Staubli VAL3: CMS_Module.dtx

bool bDoAirex = true
bool bGlueGlass
public dio doJ206_EtherCAT_Box_1__CPX_FB37__Q0 = {link=J206_EtherCAT\Box_1_(CPX-FB37)\%Q0}
public dio doJ206_EtherCAT_Box_1__CPX_FB37__Q1 = {link=J206_EtherCAT\Box_1_(CPX-FB37)\%Q1}
public dio doJ206_EtherCAT_Box_1__CPX_FB37__Q10 = {link=J206_EtherCAT\Box_1_(CPX-FB37)\%Q10}
public dio doJ206_EtherCAT_Box_1__CPX_FB37__Q11 = {link=J206_EtherCAT\Box_1_(CPX-FB37)\%Q11}
public dio doJ206_EtherCAT_Box_1__CPX_FB37__Q12 = {link=J206_EtherCAT\Box_1_(CPX-FB37)\%Q12}
public dio doJ206_EtherCAT_Box_1__CPX_FB37__Q13 = {link=J206_EtherCAT\Box_1_(CPX-FB37)\%Q13}
public dio doJ206_EtherCAT_Box_1__CPX_FB37__Q14 = {link=J206_EtherCAT\Box_1_(CPX-FB37)\%Q14}
public dio doJ206_EtherCAT_Box_1__CPX_FB37__Q15 = {link=J206_EtherCAT\Box_1_(CPX-FB37)\%Q15}
public dio doJ206_EtherCAT_Box_1__CPX_FB37__Q16 = {link=J206_EtherCAT\Box_1_(CPX-FB37)\%Q16}
public dio doJ206_EtherCAT_Box_1__CPX_FB37__Q17 = {link=J206_EtherCAT\Box_1_(CPX-FB37)\%Q17}
public dio doJ206_EtherCAT_Box_1__CPX_FB37__Q18 = {link=J206_EtherCAT\Box_1_(CPX-FB37)\%Q18}
public dio doJ206_EtherCAT_Box_1__CPX_FB37__Q19 = {link=J206_EtherCAT\Box_1_(CPX-FB37)\%Q19}
public dio doJ206_EtherCAT_Box_1__CPX_FB37__Q2 = {link=J206_EtherCAT\Box_1_(CPX-FB37)\%Q2}
public dio doJ206_EtherCAT_Box_1__CPX_FB37__Q20 = {link=J206_EtherCAT\Box_1_(CPX-FB37)\%Q20}
public dio doJ206_EtherCAT_Box_1__CPX_FB37__Q21 = {link=J206_EtherCAT\Box_1_(CPX-FB37)\%Q21}
public dio doJ206_EtherCAT_Box_1__CPX_FB37__Q22 = {link=J206_EtherCAT\Box_1_(CPX-FB37)\%Q22}
public dio doJ206_EtherCAT_Box_1__CPX_FB37__Q23 = {link=J206_EtherCAT\Box_1_(CPX-FB37)\%Q23}
public dio doJ206_EtherCAT_Box_1__CPX_FB37__Q24 = {link=J206_EtherCAT\Box_1_(CPX-FB37)\%Q24}
public dio doJ206_EtherCAT_Box_1__CPX_FB37__Q25 = {link=J206_EtherCAT\Box_1_(CPX-FB37)\%Q25}
public dio doJ206_EtherCAT_Box_1__CPX_FB37__Q26 = {link=J206_EtherCAT\Box_1_(CPX-FB37)\%Q26}
public dio doJ206_EtherCAT_Box_1__CPX_FB37__Q27 = {link=J206_EtherCAT\Box_1_(CPX-FB37)\%Q27}
public dio doJ206_EtherCAT_Box_1__CPX_FB37__Q28 = {link=J206_EtherCAT\Box_1_(CPX-FB37)\%Q28}
public dio doJ206_EtherCAT_Box_1__CPX_FB37__Q29 = {link=J206_EtherCAT\Box_1_(CPX-FB37)\%Q29}
public dio doJ206_EtherCAT_Box_1__CPX_FB37__Q3 = {link=J206_EtherCAT\Box_1_(CPX-FB37)\%Q3}
public dio doJ206_EtherCAT_Box_1__CPX_FB37__Q30 = {link=J206_EtherCAT\Box_1_(CPX-FB37)\%Q30}
public dio doJ206_EtherCAT_Box_1__CPX_FB37__Q31 = {link=J206_EtherCAT\Box_1_(CPX-FB37)\%Q31}
public dio doJ206_EtherCAT_Box_1__CPX_FB37__Q4 = {link=J206_EtherCAT\Box_1_(CPX-FB37)\%Q4}
public dio doJ206_EtherCAT_Box_1__CPX_FB37__Q5 = {link=J206_EtherCAT\Box_1_(CPX-FB37)\%Q5}
public dio doJ206_EtherCAT_Box_1__CPX_FB37__Q6 = {link=J206_EtherCAT\Box_1_(CPX-FB37)\%Q6}
public dio doJ206_EtherCAT_Box_1__CPX_FB37__Q7 = {link=J206_EtherCAT\Box_1_(CPX-FB37)\%Q7}
public dio doJ206_EtherCAT_Box_1__CPX_FB37__Q8 = {link=J206_EtherCAT\Box_1_(CPX-FB37)\%Q8}
public dio doJ206_EtherCAT_Box_1__CPX_FB37__Q9 = {link=J206_EtherCAT\Box_1_(CPX-FB37)\%Q9}
public dio switchMagnet = {link=FastIO\fOut0}
public dio switchVac0 = {link=ValveIO\valve1}
public dio switchVac1 = {link=ValveIO\valve2}
frame fPalette = {x=-254.28, y=175.62, z=30, rz=0.110016, fatherId=world[0]}
jointRs jInitialPosition = {j1=50, j2=50, j3=80, j4=15}
jointRs jRestPosition = {j1=70, j2=40, j3=80, j4=10}
mdesc mFast = {accel=2, vel=50, decel=2, tmax=60, rmax=60, leave=100}
mdesc mNomSpeed = {accel=5, vel=20, decel=5, tmax=9999, rmax=9999}
mdesc mSlow = {accel=5, vel=20, decel=5, tmax=99, rmax=99, leave=25, reach=25}
num airexValve[6]
  [0] = 12
  [1] = 6
  [3] = 13
  [4] = 7
  [5] = 1
num hdiValve[6]
  [0] = 14
  [1] = 8
  [2] = 2
  [3] = 16
  [4] = 10
  [5] = 4
num nError
num sensorValve[6]
  [0] = 15
  [1] = 9
  [2] = 3
  [3] = 17
  [4] = 11
  [5] = 5
num statusValves[32]
  [0] = 1
  [1] = 1
  [2] = 1
  [3] = 1
  [4] = 1
  [5] = 1
  [6] = 1
  [7] = 1
  [8] = 1
  [9] = 1
  [10] = 1
  [11] = 1
  [12] = 1
  [13] = 1
  [14] = 1
  [15] = 1
  [16] = 1
  [17] = 1
  [18] = 1
  [19] = 1
  [20] = 1
  [21] = 1
  [22] = 1
  [23] = 1
  [24] = 1
  [25] = 1
  [26] = 1
  [27] = 1
  [28] = 1
  [29] = 1
  [30] = 1
  [31] = 1
num waitGlue = 3
num waitShort = 1
pointRs airexFinal[6]
  [0] = {x=58.9, y=184.625, z=-97.69, rx=180, fatherId=fPalette[0]}
  [1] = {x=133.9, y=184.625, z=-97.69, rx=180, fatherId=fPalette[0]}
  [2] = {x=208.9, y=184.625, z=-97.69, rx=180, fatherId=fPalette[0]}
  [3] = {x=58.9, y=314.625, z=-97.69, rx=180, fatherId=fPalette[0]}
  [4] = {x=133.9, y=314.625, z=-97.69, rx=180, fatherId=fPalette[0]}
  [5] = {x=208.9, y=314.625, z=-97.69, rx=180, fatherId=fPalette[0]}
pointRs airexGlueStampEnd = {x=466.48, y=113.596594, z=-96.5, rx=180, ry=6.951996E-15, rz=0.0536958, fatherId=fPalette[0]}
pointRs airexGlueStampHome = {x=496, y=54, z=-97.69, rx=180, fatherId=fPalette[0]}
pointRs airexInitial[6]
  [0] = {x=59, y=114, z=-97.69, rx=180, fatherId=fPalette[0]}
  [1] = {x=134, y=114, z=-97.69, rx=180, fatherId=fPalette[0]}
  [2] = {x=209, y=114, z=-97.69, rx=180, fatherId=fPalette[0]}
  [3] = {x=59, y=144, z=-97.69, rx=180, fatherId=fPalette[0]}
  [4] = {x=134, y=144, z=-97.69, rx=180, fatherId=fPalette[0]}
  [5] = {x=209, y=144, z=-97.69, rx=180, fatherId=fPalette[0]}
pointRs chuck1[6]
  [0] = {x=59, y=39, z=-97.69, rx=180, fatherId=fPalette[0]}
  [1] = {x=134, y=39, z=-97.69, rx=180, fatherId=fPalette[0]}
  [2] = {x=209, y=39, z=-97.69, rx=180, fatherId=fPalette[0]}
  [3] = {x=59, y=79, z=-97.69, rx=180, fatherId=fPalette[0]}
  [4] = {x=134, y=79, z=-97.69, rx=180, fatherId=fPalette[0]}
  [5] = {x=209, y=79, z=-97.69, rx=180, fatherId=fPalette[0]}
pointRs chuck2[6]
  [0] = {x=291, y=54, z=-97.69, rx=180, fatherId=fPalette[0]}
  [1] = {x=361, y=54, z=-97.69, rx=180, fatherId=fPalette[0]}
  [2] = {x=291, y=119, z=-97.69, rx=180, fatherId=fPalette[0]}
  [3] = {x=361, y=119, z=-97.69, rx=180, fatherId=fPalette[0]}
  [4] = {x=291, y=184, z=-97.69, rx=180, fatherId=fPalette[0]}
  [5] = {x=361, y=184, z=-97.69, rx=180, fatherId=fPalette[0]}
pointRs gluePickPoint[6]
  [0] = {x=310, y=-15.8, z=-62.5, rx=180, ry=6.952208E-15, fatherId=world[0]}
  [1] = {x=310, y=17.2, z=-62.5, rx=180, fatherId=world[0]}
  [2] = {x=340, y=-15.8, z=-62.5, rx=180, fatherId=world[0]}
  [3] = {x=340, y=17.2, z=-62.5, rx=180, fatherId=world[0]}
  [4] = {x=370, y=-15.8, z=-62.5, rx=180, fatherId=world[0]}
  [5] = {x=370, y=17.2, z=-62.5, rx=180, fatherId=world[0]}
pointRs hdiFinal[6]
  [0] = {x=59, y=249, z=-97.69, rx=180, fatherId=fPalette[0]}
  [1] = {x=134, y=249, z=-97.69, rx=180, fatherId=fPalette[0]}
  [2] = {x=209, y=249, z=-97.69, rx=180, fatherId=fPalette[0]}
  [3] = {x=59, y=379, z=-97.69, rx=180, fatherId=fPalette[0]}
  [4] = {x=134, y=379, z=-97.69, rx=180, fatherId=fPalette[0]}
  [5] = {x=209, y=379, z=-97.69, rx=180, fatherId=fPalette[0]}
pointRs pBasisRs = {x=-45.372705, y=215.0412411, z=72.706789, rx=180, ry=6.952541E-15, rz=0.0207374, fatherId=world[0]}
pointRs pFrameUrsprung = {x=-254.28, y=175.62, z=30, fatherId=world[0]}
pointRs pFrameX = {x=271.72, y=176.63, z=30, fatherId=world[0]}
pointRs pFrameY = {x=-255.12, y=613.62, z=30, fatherId=world[0]}
string colorOff = "beige"
string colorOn = "darkgreen"
string colorValveButton[32]
  [0] = "darkgreen"
  [1] = "darkgreen"
  [2] = "darkgreen"
  [3] = "darkgreen"
  [4] = "darkgreen"
  [5] = "darkgreen"
  [6] = "darkgreen"
  [7] = "darkgreen"
  [8] = "darkgreen"
  [9] = "darkgreen"
  [10] = "darkgreen"
  [11] = "darkgreen"
  [12] = "darkgreen"
  [13] = "darkgreen"
  [14] = "darkgreen"
  [15] = "darkgreen"
  [16] = "darkgreen"
  [17] = "darkgreen"
  [18] = "darkgreen"
  [19] = "darkgreen"
  [20] = "darkgreen"
  [21] = "darkgreen"
  [22] = "darkgreen"
  [23] = "darkgreen"
  [24] = "darkgreen"
  [25] = "darkgreen"
  [26] = "darkgreen"
  [27] = "darkgreen"
  [28] = "darkgreen"
  [29] = "darkgreen"
  [30] = "darkgreen"
  [31] = "darkgreen"
public tool tTool = {z=70, rz=-97.72, fatherId=flange[0]}
trsf trApproach = {z=-20}
trsf trStamp = {z=-7}
trsf trZsafe = {z=-80}
string colorVacuumStatus1
string statusDoAirex
string colorGray
string colorRunning
string colorCleanupChuck1
string statusCleanupChuck1
mdesc mVerySlow = {accel=2, vel=5, decel=2, tmax=5, rmax=5, leave=10, reach=10}
string statusDoModules
string statusCleanupChuck2
string colorCleanupChuck2
bool bDoModules
pointRs gluePickPoint2[6]
  [0] = {x=330, y=-25, z=-62.5, rx=180, ry=6.952208E-15, fatherId=world[0]}
  [1] = {x=330, y=25, z=-62.5, rx=180, fatherId=world[0]}
  [2] = {x=380, y=-25, z=-62.5, rx=180, fatherId=world[0]}
  [3] = {x=380, y=25, z=-62.5, rx=180, fatherId=world[0]}
  [4] = {x=430, y=-25, z=-62.5, rx=180, fatherId=world[0]}
  [5] = {x=430, y=25, z=-62.5, rx=180, fatherId=world[0]}
pointRs moduleGlueStampHome = {x=436, y=54, z=-97.69, rx=180, ry=6.951996E-15, fatherId=fPalette[0]}
pointRs moduleGlueStampEnd = {x=466.48, y=156.596594, z=-96.5, rx=180, ry=6.951996E-15, rz=0.0536958, fatherId=fPalette[0]}
mdesc mExtremelySlow = {accel=0.05, vel=0.05, decel=0.05, tmax=0.04, rmax=0.04, leave=1, reach=1}
pointRs glueFirstPoint[4]
  [0] = {x=280, y=-25, z=-62.5, rx=180, ry=6.952208E-15, fatherId=world[0]}
  [1] = {x=280, y=25, z=-62.5, rx=180, fatherId=world[0]}
  [2] = {x=280, y=-5, z=-62.5, rx=180, fatherId=world[0]}
  [3] = {x=280, y=5, z=-62.5, rx=180, fatherId=world[0]}
trsf trZclose = {z=-10}
bool bSelectItem
bool bSelectedItems[6]
bool bSkipGlue
string colorError
string strStatus
trsf trZero
pointRs pSomewhere = {x=300, y=200, fatherId=world[0]}
trsf trPressTwo = {z=2}
trsf trUpTwo = {z=-8}
jointRs jPosition
string sPosition
bool bCleanup
num speedFactor
mdesc mSpeedArray[10]
  [0] = {accel=0.05, vel=0.05, decel=0.05, tmax=0.04, rmax=0.04, leave=1, reach=1}
  [1] = {accel=0.5, vel=0.5, decel=0.5, tmax=1, rmax=1, leave=2, reach=2}
  [2] = {accel=1, vel=1, decel=1, tmax=2, rmax=2, leave=2, reach=2}
  [3] = {accel=2, vel=2, decel=2, tmax=5, rmax=5, leave=5, reach=5}
  [4] = {accel=4, vel=7, decel=4, tmax=10, rmax=10, leave=10, reach=10}
  [5] = {accel=5, vel=10, decel=5, tmax=15, rmax=15, leave=20, reach=10}
  [6] = {accel=6, vel=15, decel=6, tmax=20, rmax=20, leave=20, reach=10}
  [7] = {accel=8, vel=20, decel=8, tmax=30, rmax=30, leave=40, reach=20}
  [8] = {accel=10, vel=25, decel=10, tmax=60, rmax=60, leave=40, reach=20}
  [9] = {accel=15, vel=35, decel=15, tmax=60, rmax=60, leave=80, reach=40}
trsf trDownTwo = {z=-2}
trsf trUpThree = {z=-9}
trsf trZverySafe = {z=-90}
string version
public sio sioSockets_server = {link=Socket\server}
string sReceiveMsg
string sSendMsg
public sio sioSockets_client = {link=Socket\client}
bool bGoRemote
string strTCPIP
bool bSockets
pointRs pGoRemoteTarget = {fatherId=fPalette[0]}
bool bEndProgram
pointRs parkEndPoint = {x=530, y=25, z=-62.5, rx=180, fatherId=world[0]}
trsf trXYZero
string sMovementID
trsf trPressOne = {z=1}
trsf trOne = {z=-1}
mdesc mVeryFast = {accel=10, vel=60, decel=10, tmax=9999, rmax=9999, leave=100}
trsf trXYstampOffset
trsf trXYCorrection1 = {x=0.09}
trsf trXYCorrectionHDI = {x=0.09}
pointRs glassInitial[6]
  [0] = {x=58.9, y=183.9, z=-97.69, rx=180, fatherId=fPalette[0]}
  [1] = {x=133.9, y=183.9, z=-97.69, rx=180, fatherId=fPalette[0]}
  [2] = {x=208.9, y=183.9, z=-97.69, rx=180, fatherId=fPalette[0]}
  [3] = {x=58.9, y=313.9, z=-97.69, rx=180, fatherId=fPalette[0]}
  [4] = {x=133.9, y=313.9, z=-97.69, rx=180, fatherId=fPalette[0]}
  [5] = {x=208.9, y=313.9, z=-97.69, rx=180, fatherId=fPalette[0]}
mdesc mSmooth = {accel=5, vel=20, decel=5, tmax=99, rmax=99, leave=100, blend=cartesian}
trsf trStampHDI = {z=-6}
pointRs gluePreApplicationPoint[4]
  [0] = {x=280, y=-90, z=-62.5, rx=180, ry=6.952208E-15, fatherId=world[0]}
  [1] = {x=280, y=90, z=-62.5, rx=180, fatherId=world[0]}
  [2] = {x=310, y=-90, z=-62.5, rx=180, fatherId=world[0]}
  [3] = {x=310, y=90, z=-62.5, rx=180, fatherId=world[0]}
